FUNCTION alg_s_Hinitialized : BOOL
VAR_INPUT
	state: STATE;
END_VAR

alg_s_Hinitialized := (state.dvar_M_HardwareMap) = (elit_initialized);

END_FUNCTION

(* stored: Version 1.1.0.1, ProductVersion 3.1.4022.18
   POU alg_s_Hinitialized: Id {1fa27bed-2c50-4dbe-957c-f3a652bfcad5}, SpecialFunc None *)
